(* IEC 61131-3 sources: programs/VI-54/VI-54_20171205/VI-54_20171205/Stations/Screen/LseClass170718/Class/TCPComReceive, 1 file *)

(* ---- TCPComReceive.st ---- *)
(*!
<Class
	Name               = "TCPComReceive"
	Revision           = "1.0"
	RealtimeTask       = "false"
	CyclicTask         = "false"
	BackgroundTask     = "false"
	Sigmatek           = "true"
	OSInterface        = "false"
	HighPriority       = "false"
	Automatic          = "false"
	UpdateMode         = "Prescan"
	SharedCommandTable = "true"
	Objectsize         = "(600,240)"
	Comment            = "Receiving data via communication class.">
	<Channels>
		<Server Name="ClassSvr" Visualized="false" Initialize="false" WriteProtected="true" Retentive="false"/>
		<Server Name="ID_Source" Visualized="false" Initialize="true" WriteProtected="true" Retentive="false" Comment="Source communication id number."/>
		<Server Name="sRecvCnt" Visualized="false" Initialize="false" WriteProtected="false" Retentive="false" Comment="Counter for received data blocks."/>
		<Client Name="toDataManager" Required="true" Internal="false" Comment="Connection to communication data manager."/>
	</Channels>
	<RevDoku>
		<Owner Company="Sigmatek GmbH &amp; Co KG" Author="LeiChr"/>
		<Dokumentation Revision="1.0" Date="2015-07-30" Author="LeiChr" Company="Sigmatek GmbH &amp; Co KG" Description="Initial library version"/>
	</RevDoku>
</Class>
*)
TCPComReceive : CLASS
  //Servers:
	ClassSvr 	: SvrChCmd_DINT;
	ID_Source 	: SvrCh_DINT;
	sRecvCnt 	: SvrCh_DINT;
  //Clients:
	toDataManager 	: CltChCmd_DataManager;
  //Variables:
  //Functions:

	FUNCTION VIRTUAL GLOBAL Init;
				//! <Function Comment="Is called whenever data is received. Overwrite this method to process data. &#13;&#10;NOTE: I the optional CMD parameter is used when sending, the method CallBackReciverCMD() has to be used for receiving in order to correctly receive the CMD parameter." Name="CallBackReceiver"/>
	FUNCTION VIRTUAL GLOBAL CallBackReceiver
		VAR_INPUT
			DestinationID 	: DINT;
			SourceID 	: DINT;
			size 	: UDINT;
			pdata 	: ^USINT;
		END_VAR
		VAR_OUTPUT
			retcode 	: BOOL;			//! <Variable Comment="TRUE .. erfolgreich Empfangen .._MNG_Recived &#13;&#10;FALSE.. Fehler beim Empfangen .._MNG_GlobalReciveError" Name="CallBackReceiver.retcode"/>
		END_VAR;
				//! <Function Comment="Overwrite this method in order to receive messages including the optional CMD parameter." Name="CallBackReciverCMD"/>
	FUNCTION VIRTUAL GLOBAL CallBackReciverCMD
		VAR_INPUT
			DestinationID 	: DINT;
			SourceID 	: DINT;
			size 	: UDINT;
			pdata 	: ^USINT;
			OptCMD 	: USINT;
		END_VAR
		VAR_OUTPUT
			retcode 	: BOOL;
		END_VAR;
  //Tables:
	FUNCTION @STD
		VAR_OUTPUT
			ret_code	: CONFSTATES;
		END_VAR;
	FUNCTION GLOBAL TAB @CT_;
END_CLASS;

#pragma usingLtd DataManager

// ********************************************************************
// Prototype of callbackmethod
// ********************************************************************
// ********************************************************************
FUNCTION GLOBAL CallBackReceiverFnc_TCPComReceive
	VAR_INPUT
		pthis 	: ^void;
		DestinationID 	: DINT;
		SourceID 	: DINT;
		size 	: UDINT;
		pdata 	: ^USINT;
	END_VAR
  var_output
    retcode : bool;
  end_var

  retcode := pthis$^TCPComReceive^.CallBackReceiver(DestinationID, SourceID, size, pdata);
  pthis$^TCPComReceive^.sRecvCnt +=1;

END_FUNCTION

// ********************************************************************
// init method
// connect the receiver do datamanager
// ********************************************************************
// ********************************************************************
FUNCTION VIRTUAL GLOBAL TCPComReceive::Init

  if _FirstScan then
     // Als Empfangsklasse anmelden
    if toDataManager.ConnectReciver(udID      := ID_Source,
                                    pThis     := this,
                                    pCallback := #CallBackReceiverFnc_TCPComReceive()) <> 1 then

      TRACE("TCPComSend_Data::Init(): Fehler beim Anmelden als Empfangsklasse");
      ClassSvr := ERROR;
    end_if;

  end_if;

END_FUNCTION

// ********************************************************************
// callbackmethod of receiver
// ********************************************************************
// ********************************************************************
FUNCTION VIRTUAL GLOBAL TCPComReceive::CallBackReceiver
	VAR_INPUT
		DestinationID 	: DINT;
		SourceID 	: DINT;
		size 	: UDINT;
		pdata 	: ^USINT;
	END_VAR
	VAR_OUTPUT
		retcode 	: BOOL;
	END_VAR

  retcode := CallBackReciverCMD(DestinationID:=(DestinationID AND 16#00FFFFFF),
                                SourceID:=SourceID,
                                size:=size,
                                pdata:=pdata,
                                OptCMD:= to_usint((DestinationID$udint AND 16#FF000000) shr 24)  );

END_FUNCTION

// ********************************************************************
// callbackmethod to handle the data
// ********************************************************************
// ********************************************************************
FUNCTION VIRTUAL GLOBAL TCPComReceive::CallBackReciverCMD
#pragma warning(disable:73);
  VAR_INPUT
		DestinationID 	: DINT;
		SourceID 	: DINT;
		size 	: UDINT;
		pdata 	: ^USINT;
		OptCMD 	: USINT;
	END_VAR
#pragma warning(default:73);

	VAR_OUTPUT
		retcode 	: BOOL;
	END_VAR

  // received data
  retcode := TRUE;

END_FUNCTION
